Staubli VAL3: onF6Event.pgx

program onF6Event()
  local string l_sItem
begin
  // look if the bButton is enable

end
